FUNCTION_BLOCK Decoder (* Basic Function Block Type *)
  (* Standard: 61499-2 *)
  (* Version 0.0, 5/5/2019, erik, nxtControl GmbH, Template *)
  PACKAGE Main;
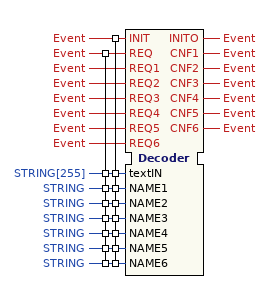
  EVENT_INPUT
    INIT WITH textIN, NAME1, NAME2, NAME3, NAME4, NAME5, NAME6; (* Initialization Request *)
    REQ WITH textIN, NAME1, NAME2, NAME3, NAME4, NAME5, NAME6; (* Normal Execution Request *)
    REQ1;
    REQ2;
    REQ3;
    REQ4;
    REQ5;
    REQ6;
  END_EVENT
  EVENT_OUTPUT
    INITO; (* Initialization Confirm *)
    CNF1; (* Execution Confirmation *)
    CNF2;
    CNF3;
    CNF4;
    CNF5;
    CNF6;
  END_EVENT
  VAR_INPUT
    textIN : STRING[255];
    NAME1 : STRING; (* Input event qualifier *)
    NAME2 : STRING;
    NAME3 : STRING;
    NAME4 : STRING;
    NAME5 : STRING;
    NAME6 : STRING;
  END_VAR
  VAR
    Internal_var1 : DINT;
  END_VAR
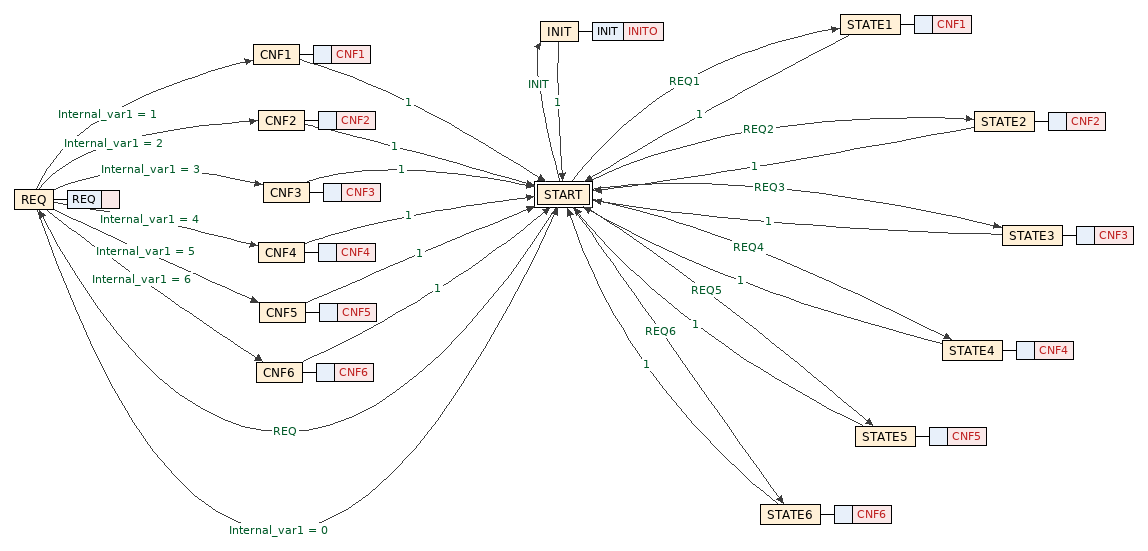
  EC_STATES
    START; (* Initial State *)
    INIT : INIT -> INITO; (* Initialization *)
    REQ : REQ; (* Normal execution *)
    CNF1 : -> CNF1;
    CNF2 : -> CNF2;
    CNF3 : -> CNF3;
    CNF4 : -> CNF4;
    CNF5 : -> CNF5;
    CNF6 : -> CNF6;
    STATE1 : -> CNF1;
    STATE2 : -> CNF2;
    STATE3 : -> CNF3;
    STATE4 : -> CNF4;
    STATE5 : -> CNF5;
    STATE6 : -> CNF6;
  END_STATES
  EC_TRANSITIONS
    START TO INIT := INIT;
    INIT TO START := 1;
    START TO REQ := REQ;
    REQ TO CNF1 := Internal_var1 = 1;
    REQ TO CNF2 := Internal_var1 = 2;
    REQ TO CNF3 := Internal_var1 = 3;
    REQ TO CNF4 := Internal_var1 = 4;
    REQ TO CNF5 := Internal_var1 = 5;
    REQ TO CNF6 := Internal_var1 = 6;
    CNF6 TO START := 1;
    CNF2 TO START := 1;
    CNF1 TO START := 1;
    CNF3 TO START := 1;
    CNF4 TO START := 1;
    CNF5 TO START := 1;
    START TO STATE1 := REQ1;
    START TO STATE2 := REQ2;
    START TO STATE3 := REQ3;
    START TO STATE4 := REQ4;
    START TO STATE5 := REQ5;
    START TO STATE6 := REQ6;
    STATE6 TO START := 1;
    STATE5 TO START := 1;
    STATE4 TO START := 1;
    STATE3 TO START := 1;
    STATE2 TO START := 1;
    STATE1 TO START := 1;
    REQ TO START := Internal_var1 = 0;
  END_TRANSITIONS
  ALGORITHM INIT IN ST: (* Initialization algorithm *)
;
Internal_var1 := 0;
  END_ALGORITHM
  ALGORITHM REQ IN ST: (* Normally executed algorithm *)
;
  END_ALGORITHM
END_FUNCTION_BLOCK
